FUNCTION_BLOCK FB_MessageQueue
VAR CONSTANT
	COMMAND_QUEUE_BUFFER_SIZE :UDINT := 5;
END_VAR
VAR_OUTPUT
END_VAR
VAR
	_usage:	UDINT;
	_write_index : UDINT := 1;
	_read_index : UDINT := 1;
	_queue_size:	UDINT := COMMAND_QUEUE_BUFFER_SIZE;
	queue_buffer:	ARRAY [1..COMMAND_QUEUE_BUFFER_SIZE] OF ST_CommandContainer;
END_VAR

PROPERTY full : BOOL
GET
full :=  _usage >= COMMAND_QUEUE_BUFFER_SIZE;
END_GET
END_PROPERTY

METHOD get : REFERENCE TO ST_CommandContainer
VAR_INPUT
END_VAR
IF _usage = 0 THEN
	get REF= 0;
	RETURN;
END_IF

get REF= queue_buffer[_read_index];

_usage := _usage - 1;

IF COMMAND_QUEUE_BUFFER_SIZE > _read_index THEN
	_read_index := _read_index + 1;
ELSE
	_read_index := 1;
END_IF
END_METHOD

METHOD put : BOOL
VAR_INPUT
	sender : ITF_Sender;
	receiver : ITF_Receiver;
END_VAR
IF _usage >= COMMAND_QUEUE_BUFFER_SIZE THEN
	put := FALSE;
ELSE
	queue_buffer[_write_index].sender := sender;
	queue_buffer[_write_index].receiver := receiver;
	_usage := _usage + 1;
	IF COMMAND_QUEUE_BUFFER_SIZE > _write_index THEN
		_write_index := _write_index + 1;
	ELSE
		_write_index := 1;
	END_IF
	put := TRUE;
END_IF
END_METHOD

PROPERTY usage : UDINT
GET
usage := _usage;
END_GET
END_PROPERTY

END_FUNCTION_BLOCK

(* stored: Version 1.1.0.1, ProductVersion 3.1.4024.15
   POU FB_MessageQueue: Id {a7278202-b575-4577-a458-ddcec29012ba}, SpecialFunc None
   Property full: Id {e3de9c67-ef8c-4885-b0d0-c9c6d8211ff9}
   Get Get: Id {f87d1f5c-efdd-40b1-a1b7-dd2f20e9ba27}
   Method get: Id {04898b93-8bb3-4ba5-8551-03f4d77e5729}
   Method put: Id {93203208-f677-42c4-9276-d0f7d8d17596}
   Property usage: Id {968b256f-6a05-45a5-bf92-8b94f3403299}
   Get Get: Id {aed42d38-7947-47bf-86fe-81eeea8e9812} *)
